INTERFACE I_WaterController

METHOD GetDuration : TIME
VAR_INPUT
	stWash : REFERENCE TO ST_Wash;
END_VAR
END_METHOD

METHOD StartDrain : BOOL
VAR_INPUT
END_VAR
END_METHOD

METHOD StartFill : BOOL
VAR_INPUT
END_VAR
END_METHOD

METHOD Stop : BOOL
VAR_INPUT
END_VAR
END_METHOD

END_INTERFACE

(* stored: Version 1.1.0.1, ProductVersion 3.1.4024.16
   Itf I_WaterController: Id {012b58e9-6e55-44d0-9c5b-8788f5458c55}
   Method GetDuration: Id {b3a329eb-3e42-46bb-a615-ebad9e5af793}
   Method StartDrain: Id {25053972-740d-4e05-b8dd-5a7435364f92}
   Method StartFill: Id {47c7ab24-b7a8-4e8f-b304-04490c99e0a1}
   Method Stop: Id {57200dc2-4fdc-418d-afba-84f2bfe13a2b} *)
